# EPICS autosave request: evtApp/Db/ADEmergentVision_settings.req
file "ADBase_settings.req",       P=$(P),  R=cam1:
